// TIA Portal V15.1 export
// export: Created 2024-05-17T05:38:15.9522421Z, ExportSetting WithDefaults, DisplayName Totally Integrated Automation Portal, DisplayVersion V15.1 Update 5, DisplayName TIA Portal Openness, DisplayVersion V15.1 Update 5, DisplayName SINAMICS Startdrive Advanced, DisplayVersion V15.1, DisplayName G130, G150, S120, S150, SINAMICS MV, S210, DisplayVersion V15.1, DisplayName G110M, G120, G120C, G120D, G120P, DisplayVersion V15.1, DisplayName STEP 7 Professional, DisplayVersion V15.1 Update 5, DisplayName STEP 7 Safety, DisplayVersion V15.1, DisplayName WinCC Professional, DisplayVersion V15.1 Update 5, DisplayName SIMATIC Visualization Architect, DisplayVersion V15.1
DATA_BLOCK "_209210ZM01DataHandling"   // DB304
{ S7_Optimized_Access := 'FALSE' }
AUTHOR : VCC
VERSION : 0.1
// stored: AutoNumber false, DBAccessibleFromOPCUA true, IsOnlyStoredInLoadMemory false, IsWriteProtectedInAS false
   VAR RETAIN
      AC_209210NCB01VIDSMasterAlarm { ExternalAccessible := 'False'; ExternalVisible := 'False'; ExternalWritable := 'False'} : Bool;   // VIDS 209210NCB01 - Master Alarm
      AC_209210NCB01VIDSRFIDAlarm { ExternalAccessible := 'False'; ExternalVisible := 'False'; ExternalWritable := 'False'} : Bool;   // VIDS 209210NCB01 - RFID Alarm
      AC_209210NCB01VIDSTrackingAlarm { ExternalAccessible := 'False'; ExternalVisible := 'False'; ExternalWritable := 'False'} : Bool;   // VIDS 209210NCB01 - Tracking Alarm
      AC_209210NCB02VIDSMasterAlarm { ExternalAccessible := 'False'; ExternalVisible := 'False'; ExternalWritable := 'False'} : Bool;   // VIDS 209210NCB02 - Master Alarm
      AC_209210NCB02VIDSRFIDAlarm { ExternalAccessible := 'False'; ExternalVisible := 'False'; ExternalWritable := 'False'} : Bool;   // VIDS 209210NCB02 - RFID Alarm
      AC_209210NCB02VIDSQualityRequestAlarm { ExternalAccessible := 'False'; ExternalVisible := 'False'; ExternalWritable := 'False'} : Bool;   // VIDS 209210NCB02 - Quality Request Alarm
      AC_209210NCB02VIDSTrackingAlarm { ExternalAccessible := 'False'; ExternalVisible := 'False'; ExternalWritable := 'False'} : Bool;   // VIDS 209210NCB02 - Tracking Alarm
      H_HMICmd : Word;   // Commands from HMI
      H_Anim : Word;   // Animation
      H_DBnr : Int;   // DB number
      H_209210NCB01TagSequenceIAnim : Word;   // Icon Animation
      H_209210NCB02TagSequenceIAnim : Word;   // Icon Animation
      H_HMI : Struct   // HMI Animation
         "209210NCB01VIDSMaster" : "H_HMI";   // HMI Animation
         "209210NCB01VIDSRFID" : "H_HMI";   // HMI Animation
         "209210NCB01VIDSTracking" : "H_HMI";   // HMI Animation
         "209210NCB02VIDSMaster" : "H_HMI";   // HMI Animation
         "209210NCB02VIDSRFID" : "H_HMI";   // HMI Animation
         "209210NCB02VIDSQualityRequest" : "H_HMI";   // HMI Animation
         "209210NCB02VIDSTracking" : "H_HMI";   // HMI Animation
      END_STRUCT;
      H : Struct   // HMI Animation
         "209210NCB01VIDSMaster" : "H_LVIDSMaster";   // HMI Animation
         "209210NCB01VIDSRFID" : "H_LVIDSRFID";   // HMI Animation
         "209210NCB01VIDSTracking" : "H_LVIDSTrack";   // HMI Animation
         "209210NCB02VIDSMaster" : "H_LVIDSMaster";   // HMI Animation
         "209210NCB02VIDSRFID" : "H_LVIDSRFID";   // HMI Animation
         "209210NCB02VIDSQualityRequest" : "H_LVIDSQualityRequest";   // HMI Animation
         "209210NCB02VIDSTracking" : "H_LVIDSTrack";   // HMI Animation
      END_STRUCT;
      AlarmABCondition { ExternalAccessible := 'False'; ExternalVisible := 'False'; ExternalWritable := 'False'} : Bool;   // Alarm AB condition
      AlarmA { ExternalAccessible := 'False'; ExternalVisible := 'False'; ExternalWritable := 'False'} : Bool;   // Alarm A
      AlarmB { ExternalAccessible := 'False'; ExternalVisible := 'False'; ExternalWritable := 'False'} : Bool;   // Alarm B
      AlarmC { ExternalAccessible := 'False'; ExternalVisible := 'False'; ExternalWritable := 'False'} : Bool;   // Alarm C
      AlarmD { ExternalAccessible := 'False'; ExternalVisible := 'False'; ExternalWritable := 'False'} : Bool;   // Alarm D
      "209210NCB01TagSequence" { ExternalAccessible := 'False'; ExternalVisible := 'False'; ExternalWritable := 'False'} : "AlarmBits";   // Tag Sequence Alarm Bits
      "209210NCB01ReadBegin" { ExternalAccessible := 'False'; ExternalVisible := 'False'; ExternalWritable := 'False'} : Bool;   // Start Reading Body Data
      "209210NCB01BodyData" { ExternalAccessible := 'False'; ExternalVisible := 'False'; ExternalWritable := 'False'; S7_SetPoint := 'True'} : "VEMData";   // Body Data from VEMData
      "209210NCB02TagSequence" { ExternalAccessible := 'False'; ExternalVisible := 'False'; ExternalWritable := 'False'} : "AlarmBits";   // Tag Sequence Alarm Bits
      "209210NCB02ReadBegin" { ExternalAccessible := 'False'; ExternalVisible := 'False'; ExternalWritable := 'False'} : Bool;   // Start Reading Body Data
      "209210NCB02BodyData" { ExternalAccessible := 'False'; ExternalVisible := 'False'; ExternalWritable := 'False'; S7_SetPoint := 'True'} : "VEMData";   // Body Data from VEMData
      "______209210NCB01_VIDS Master______" { ExternalAccessible := 'False'; ExternalVisible := 'False'; ExternalWritable := 'False'} : Bool;   // -----------------------------------------------------------------------------------
      "209210NCB01VIDS" { ExternalAccessible := 'False'; ExternalVisible := 'False'; ExternalWritable := 'False'; S7_SetPoint := 'True'} : "VIDS";   // Internal record
      "209210NCB01VEMData" { ExternalAccessible := 'False'; ExternalVisible := 'False'; ExternalWritable := 'False'; S7_SetPoint := 'True'} : "VEMData";   // VEM Data
      "209210NCB01VEMDataChange" { ExternalAccessible := 'False'; ExternalVisible := 'False'; ExternalWritable := 'False'; S7_SetPoint := 'True'} : "VEMData";   // VEM Data Change
      "209210NCB01VEMDataValid" { ExternalAccessible := 'False'; ExternalVisible := 'False'; ExternalWritable := 'False'; S7_SetPoint := 'True'} : Bool;   // VEM Data Valid
      "209210NCB01VEMDataNotValid" { ExternalAccessible := 'False'; ExternalVisible := 'False'; ExternalWritable := 'False'; S7_SetPoint := 'True'} : Bool;   // VEM Data Not Valid
      "209210NCB01GetVEMDataBusy" { ExternalAccessible := 'False'; ExternalVisible := 'False'; ExternalWritable := 'False'; S7_SetPoint := 'True'} : Bool;   // Get VEM Data Busy
      "209210NCB01MasterStatus" { ExternalAccessible := 'False'; ExternalVisible := 'False'; ExternalWritable := 'False'; S7_SetPoint := 'True'} : Int;   // Master - Status
      "______209210NCB01_VIDS RFID______" { ExternalAccessible := 'False'; ExternalVisible := 'False'; ExternalWritable := 'False'} : Bool;   // -----------------------------------------------------------------------------------
      "209210NCB01ReadOK" { ExternalAccessible := 'False'; ExternalVisible := 'False'; ExternalWritable := 'False'; S7_SetPoint := 'True'} : Bool;   // RFID - Read OK
      "209210NCB01ReadNOK" { ExternalAccessible := 'False'; ExternalVisible := 'False'; ExternalWritable := 'False'; S7_SetPoint := 'True'} : Bool;   // RFID - Read NOK
      "209210NCB01Busy" { ExternalAccessible := 'False'; ExternalVisible := 'False'; ExternalWritable := 'False'; S7_SetPoint := 'True'} : Bool;   // RFID - Busy
      "209210NCB01Status" { ExternalAccessible := 'False'; ExternalVisible := 'False'; ExternalWritable := 'False'; S7_SetPoint := 'True'} : Int;   // RFID - Status
      "______209210NCB01_VIDS Tracking______" { ExternalAccessible := 'False'; ExternalVisible := 'False'; ExternalWritable := 'False'} : Bool;   // -----------------------------------------------------------------------------------
      "209210NCB01TrackOK" { ExternalAccessible := 'False'; ExternalVisible := 'False'; ExternalWritable := 'False'; S7_SetPoint := 'True'} : Bool;   // Track - OK
      "209210NCB01TrackNOK" { ExternalAccessible := 'False'; ExternalVisible := 'False'; ExternalWritable := 'False'; S7_SetPoint := 'True'} : Bool;   // Track - Nok
      "209210NCB01TrackBusy" { ExternalAccessible := 'False'; ExternalVisible := 'False'; ExternalWritable := 'False'; S7_SetPoint := 'True'} : Bool;   // Track - Busy
      "209210NCB01TrackStatus" { ExternalAccessible := 'False'; ExternalVisible := 'False'; ExternalWritable := 'False'; S7_SetPoint := 'True'} : Int;   // Track - Status
      "209210NCB01SpecificData" { ExternalAccessible := 'False'; ExternalVisible := 'False'; ExternalWritable := 'False'; S7_SetPoint := 'True'} : Array[0..7925] of Byte;   // Specific Data Received
      "______209210NCB02_VIDS Master______" { ExternalAccessible := 'False'; ExternalVisible := 'False'; ExternalWritable := 'False'} : Bool;   // -----------------------------------------------------------------------------------
      "209210NCB02VIDS" { ExternalAccessible := 'False'; ExternalVisible := 'False'; ExternalWritable := 'False'; S7_SetPoint := 'True'} : "VIDS";   // Internal record
      "209210NCB02VEMData" { ExternalAccessible := 'False'; ExternalVisible := 'False'; ExternalWritable := 'False'; S7_SetPoint := 'True'} : "VEMData";   // VEM Data
      "209210NCB02VEMDataChange" { ExternalAccessible := 'False'; ExternalVisible := 'False'; ExternalWritable := 'False'; S7_SetPoint := 'True'} : "VEMData";   // VEM Data Change
      "209210NCB02VEMDataValid" { ExternalAccessible := 'False'; ExternalVisible := 'False'; ExternalWritable := 'False'; S7_SetPoint := 'True'} : Bool;   // VEM Data Valid
      "209210NCB02VEMDataNotValid" { ExternalAccessible := 'False'; ExternalVisible := 'False'; ExternalWritable := 'False'; S7_SetPoint := 'True'} : Bool;   // VEM Data Not Valid
      "209210NCB02GetVEMDataBusy" { ExternalAccessible := 'False'; ExternalVisible := 'False'; ExternalWritable := 'False'; S7_SetPoint := 'True'} : Bool;   // Get VEM Data Busy
      "209210NCB02MasterStatus" { ExternalAccessible := 'False'; ExternalVisible := 'False'; ExternalWritable := 'False'; S7_SetPoint := 'True'} : Int;   // Master - Status
      "______209210NCB02_VIDS RFID______" { ExternalAccessible := 'False'; ExternalVisible := 'False'; ExternalWritable := 'False'} : Bool;   // -----------------------------------------------------------------------------------
      "209210NCB02ReadOK" { ExternalAccessible := 'False'; ExternalVisible := 'False'; ExternalWritable := 'False'; S7_SetPoint := 'True'} : Bool;   // RFID - Read OK
      "209210NCB02ReadNOK" { ExternalAccessible := 'False'; ExternalVisible := 'False'; ExternalWritable := 'False'; S7_SetPoint := 'True'} : Bool;   // RFID - Read NOK
      "209210NCB02Busy" { ExternalAccessible := 'False'; ExternalVisible := 'False'; ExternalWritable := 'False'; S7_SetPoint := 'True'} : Bool;   // RFID - Busy
      "209210NCB02Status" { ExternalAccessible := 'False'; ExternalVisible := 'False'; ExternalWritable := 'False'; S7_SetPoint := 'True'} : Int;   // RFID - Status
      "______209210NCB02_VIDS Quality Request______" { ExternalAccessible := 'False'; ExternalVisible := 'False'; ExternalWritable := 'False'} : Bool;   // -----------------------------------------------------------------------------------
      "209210NCB02Quality RequestDataValid" { ExternalAccessible := 'False'; ExternalVisible := 'False'; ExternalWritable := 'False'; S7_SetPoint := 'True'} : Bool;   // Quality Request - Data Valid
      "209210NCB02Quality RequestDataNotValid" { ExternalAccessible := 'False'; ExternalVisible := 'False'; ExternalWritable := 'False'; S7_SetPoint := 'True'} : Bool;   // Quality Request - Data Not Valid
      "209210NCB02Quality RequestBusy" { ExternalAccessible := 'False'; ExternalVisible := 'False'; ExternalWritable := 'False'; S7_SetPoint := 'True'} : Bool;   // Quality Request - Busy
      "209210NCB02Quality RequestStatus" { ExternalAccessible := 'False'; ExternalVisible := 'False'; ExternalWritable := 'False'; S7_SetPoint := 'True'} : Int;   // Quality Request - Status
      "209210NCB02Quality RequestVEMData" { ExternalAccessible := 'False'; ExternalVisible := 'False'; ExternalWritable := 'False'; S7_SetPoint := 'True'} : "VEMData";   // Quality Request - VEM Data
      "______209210NCB02_VIDS Tracking______" { ExternalAccessible := 'False'; ExternalVisible := 'False'; ExternalWritable := 'False'} : Bool;   // -----------------------------------------------------------------------------------
      "209210NCB02TrackOK" { ExternalAccessible := 'False'; ExternalVisible := 'False'; ExternalWritable := 'False'; S7_SetPoint := 'True'} : Bool;   // Track - OK
      "209210NCB02TrackNOK" { ExternalAccessible := 'False'; ExternalVisible := 'False'; ExternalWritable := 'False'; S7_SetPoint := 'True'} : Bool;   // Track - Nok
      "209210NCB02TrackBusy" { ExternalAccessible := 'False'; ExternalVisible := 'False'; ExternalWritable := 'False'; S7_SetPoint := 'True'} : Bool;   // Track - Busy
      "209210NCB02TrackStatus" { ExternalAccessible := 'False'; ExternalVisible := 'False'; ExternalWritable := 'False'; S7_SetPoint := 'True'} : Int;   // Track - Status
      "209210NCB02SpecificData" { ExternalAccessible := 'False'; ExternalVisible := 'False'; ExternalWritable := 'False'; S7_SetPoint := 'True'} : Array[0..7925] of Byte;   // Specific Data Received
   END_VAR
BEGIN
END_DATA_BLOCK
